# EPICS autosave request: ADApp/Db/firewireFeature_settings.req
$(P)$(R)$(FEATURE)
$(P)$(R)$(FEATURE)_CTRL
